// TIA Portal V20 export
TYPE "LConSMC_typeWinderInput"
// stored: Access Published
   STRUCT
      enable : Bool := FALSE;   // TRUE: Enable function block. WIth rising edge a validation of parameter is done and communication with drive is started FALSE: Disable the function block
      speedMatch : Bool := FALSE;   // TRUE: Enable web velocity setpoint ("lineAxisMotionVector"). The drive will synchronize up to web velocity using syncronization dynamics. If the velocity is reached the output "inSync" will become TRUE. FALSE: Drive will decelerate to standstill using stop dynamics
      cntrlEnable : Bool := FALSE;   // TRUE: Enable web tension control (enable torque limits, dancer position setpoint etc.)
      jogPos : Bool := FALSE;   // TRUE: Drive is jogged in positive direction (see config.dynamics.jogDynamics)
      jogNeg : Bool := FALSE;   // TRUE: Drive is jogged in negative direction (see config.dynamics.jogDynamics)
      lineAxisMotionVector : "LConSMC_typeMotionVector";   // Setpoint of the web (position/velocity/acceleration)
      lineAxisActualValues : "LConSMC_typeLineAxisActValues";   // Actual values of the web for diameter calculation. Leading value (actual or setpoint values) must be connected to the input "lineAxisMotionVector"
      additionalVelocity : LReal := 0.0;   // [m/min] / [ft/min] Additional web velocity (always enabled)
      typeOfWinder : Int;   // Definition of winding direction 0: Rewind from above 1: Rewind from below 2: Unwind from above 3: Unwind from below
      controlMode : Int := 0;   // Tension control mode 0: Dancer via speed setpoint adaption 1: Load cell via speed setpoint adaption 2: Load cell via torque limits 3: Indirect tension control 4: V-constant / Tension control mode 0: Dancer via speed setpoint adaption 1: Load cell via speed setpoint adaption 2: Load cell via torque limits 3: Indirect tension control 4: Speed setpoint relation (Draw) 5: Indirect tension control vis speed setpoint adaption
      typeOfDiameterCalc : Int;   // Type of diameter calculation 0: V/n 1: Thickness addition 2: Integral 3: External 4: WebLength 5: Position
      holdDiameter : Bool := FALSE;   // TRUE: Hold diameter calculation FALSE: Diameter calculation is active
      setDiameter : Bool := FALSE;   // TRUE: Set diameter to the value in "winderConfig.diamConfig.diameterSetValue"
      CntrlSetpoint : LReal := 0.0;   // Tension setpoint [N]/[Lbf] / Dancer position setpoint [%]
      CntrlActual : LReal := 0.0;   // Tension actual value [N]/[Lbf] / Dancer actual position [%]
      tCycle : Real := 0.0;   // [ms] Cycle time the function block is called
      winderAxis : DB_ANY;   // Winder axis
   END_STRUCT;
END_TYPE
